INTERFACE PUBLIC I_MoveRelativeBuilder EXTENDS __System.IQueryInterface

METHOD PUBLIC Acceleration : I_MoveBuilder
VAR_INPUT
	value : LREAL;
END_VAR
END_METHOD

METHOD PUBLIC BufferMode : I_MoveBuilder
VAR_INPUT
	mode : AxisBufferMode;
END_VAR
END_METHOD

METHOD PUBLIC BuildMoveAdditiveCommand : I_MoveCommand
END_METHOD

METHOD PUBLIC BuildMoveRelativeCommand : I_MoveCommand
END_METHOD

METHOD PUBLIC Deceleration : I_MoveBuilder
VAR_INPUT
	value : LREAL;
END_VAR
END_METHOD

METHOD PUBLIC Distance : I_MoveRelativeBuilder
VAR_INPUT
	value : LREAL;
END_VAR
END_METHOD

METHOD PUBLIC Jerk : I_MoveBuilder
VAR_INPUT
	value : LREAL;
END_VAR
END_METHOD

METHOD PUBLIC Velocity : I_MoveBuilder
VAR_INPUT
	value : LREAL;
END_VAR
END_METHOD

END_INTERFACE

(* stored: Version 1.1.0.1, ProductVersion 3.1.4024.12
   Itf I_MoveRelativeBuilder: Id {92bfbb92-30ca-044e-2086-373ce6e74546}
   Method Acceleration: Id {bc2fcec8-2803-0c6f-02df-3be45e1f6930}
   Method BufferMode: Id {e20fd57c-c923-043d-20d1-027baa20e4f1}
   Method BuildMoveAdditiveCommand: Id {19fe8faf-fac6-024a-1ae4-eb0d85d91941}
   Method BuildMoveRelativeCommand: Id {a7a86cde-a9a1-0ba9-3f20-8cc71c1ec9e9}
   Method Deceleration: Id {09bee452-7f5a-0fb1-1473-8c146dc19f50}
   Method Distance: Id {540dfee5-5339-0731-2f18-2e04d53bf765}
   Method Jerk: Id {deafd6ef-a4a1-06a3-26d1-2414840d5025}
   Method Velocity: Id {542cbae5-b808-01b7-1173-3727773f7285} *)
